INTERFACE I_Enable

PROPERTY Busy : bool
GET
END_GET
END_PROPERTY

METHOD Disable : BOOL
VAR_INPUT
END_VAR
END_METHOD

METHOD Enable : BOOL
VAR_INPUT
END_VAR
END_METHOD

PROPERTY Error : bool
GET
END_GET
END_PROPERTY

METHOD Parametrise : BOOL
VAR_INPUT
END_VAR
END_METHOD

METHOD RegisterAxis : BOOL
VAR_INPUT
END_VAR
END_METHOD

END_INTERFACE

(* stored: Version 1.1.0.1, ProductVersion 3.1.4024.3
   Itf I_Enable: Id {10058e29-b414-4bb7-9085-5ab6d0d16f75}
   Property Busy: Id {84941abf-4c9b-4f71-b92f-e4daa9354268}
   Get Get: Id {8ff847dc-5a97-4397-8de2-b75c26017a19}
   Method Disable: Id {348062ea-364b-4e6a-8aa9-3dc0d148c69e}
   Method Enable: Id {3a63a96a-c190-46b7-b7b2-ec404589485d}
   Property Error: Id {a1a48a46-7b62-4b8d-b3e3-561de6190465}
   Get Get: Id {e3a63eb5-3c84-42c7-93a8-9556fa9f6ced}
   Method Parametrise: Id {54194fcf-c71e-458b-be48-605a1fbea816}
   Method RegisterAxis: Id {f6d50491-a91f-448d-8ef3-593d972be9d5} *)
